FUNCTION_BLOCK FB_MotionAxisMoveAbsoluteTestDouble IMPLEMENTS I_MotionAxisMoveAbsolute
VAR
END_VAR

END_FUNCTION_BLOCK

(* stored: Version 1.1.0.1
   POU FB_MotionAxisMoveAbsoluteTestDouble: Id {265417a5-e30e-4e24-8734-206b7ae49b32}, SpecialFunc None *)
